Staubli VAL3: statistics.dtx

mdesc mNomSpeed
num nTemp
num nInput[8]
num nCopy
